RoboDK station: nfactorial.rdk

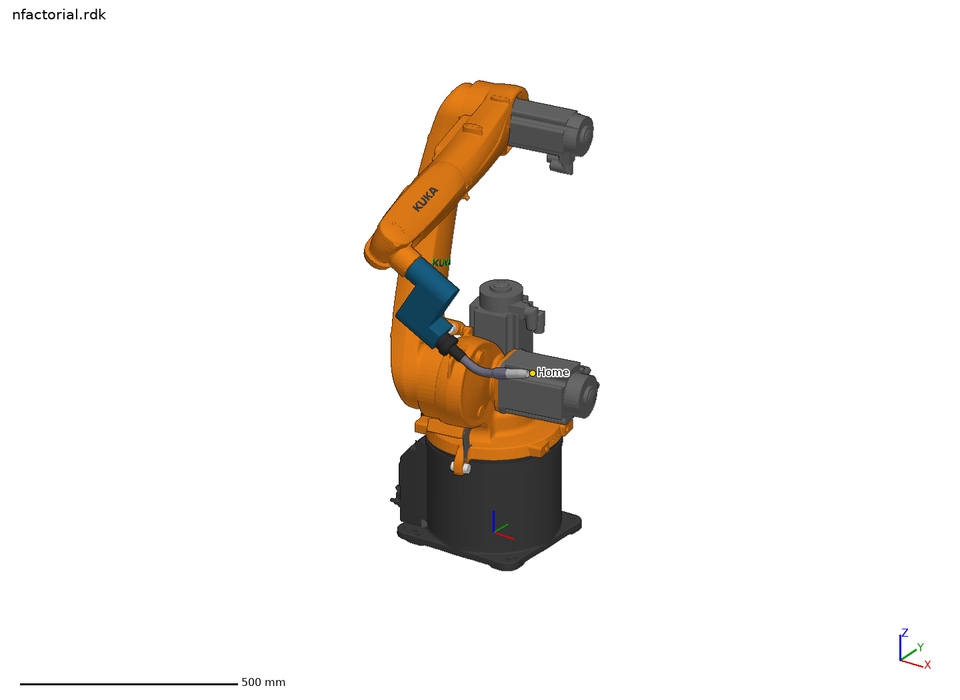
[picture v0: the station drawn from its stored meshes, robots at their saved joint values, targets as dots, program paths as lines]
Station nfactorial (saved by RoboDK 5.7.0). Poses are relative to the parent item; angles as X-Y-Z fixed-axis rotations.
Station parameters (name, value as stored): LIN64
  - frame KUKA KR 10 R1420 Base at (0, 0, 0) mm
    - robot KUKA KR 10 R1420: 6 axes, payload 10 kg, reach 1420 mm, repeatability 0.04 mm, weight 160 kg
        modified DH rows (alpha deg, a mm, theta deg, d mm): 0, 0, 0, 450; -90, 150, 0, 0; 0, 610, -90, 0; -90, 20, 0, 660; 90, 0, 0, 0; -90, 0, 180, 80
        joint limits [-170, -185, -137, -185, -120, -350] to [170, 65, 163, 185, 120, 350]; home [0, -90, 90, 0, 0, 0]; saved at [80.237, -112.594, 116.289, -58.168, 85.387, -91.774]
      - tool Weld gun, TCP at (-4, 0, 371.3) mm, rotated rx 0 ry 45 rz 0 deg, size 299.9 x 60 x 318.3 mm
    - target Home (Cartesian target) at (475.67, -523.05, 748.11) mm, rotated rx -12.12 ry -76.75 rz -163.29 deg; joints [80.237, -112.594, 116.289, -58.168, 85.387, -91.774] of KUKA KR 10 R1420
    - target Target 1 (Cartesian target) at (475.67, -523.05, 748.11) mm, rotated rx -12.12 ry -76.75 rz -163.29 deg; joints [80.237, -112.594, 116.289, -58.168, 85.387, -91.774] of KUKA KR 10 R1420
  - Python program simple (listed below)

--- Python program simple ---

